ABB RobotStudio station: Solution3Working.rspag

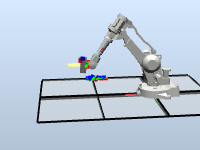
--- station ---
Station Solution3 (saved by RobotStudio 6.8.8307.1040)
Controller IRB_2400_12kg_1.55m
  mechanical unit ROB_1: IRB2400_10_150__02, 6 joints, base frame (0, 0, 0) mm
Layout (positions relative to the parent item):
  - IRB2400_10_150__02 [mechanism, from Robots\IRB2400_10_150_G_02.rslib] at (0, 0, 0) mm; joint values [0, 0.7222, 0.9922, 0, -0.9957, 0] (rad or m)
  - SickBox [smart component] at (1500, 0, 600) mm, rotated rx 0 ry -90 rz 0 deg
      properties: PointA=[1.29074548339844 0 0.569999938964844]; PointB=[1.28920959472656 0 0.6]; PointC=[1.29286682128906 0.0300000152587891 0.599999938964844]; Ax=1.29074548339844; Ay=0; Az=0.569999938964844; Bx=1.28920959472656; By=0; Bz=0.6; Cx=1.29286682128906; Cy=0.0300000152587891; Cz=0.599999938964844
      signals: AO Ax, AO Ay, AO Az, AO Bx, AO By, AO Bz, AO Cx, AO Cy, AO Cz
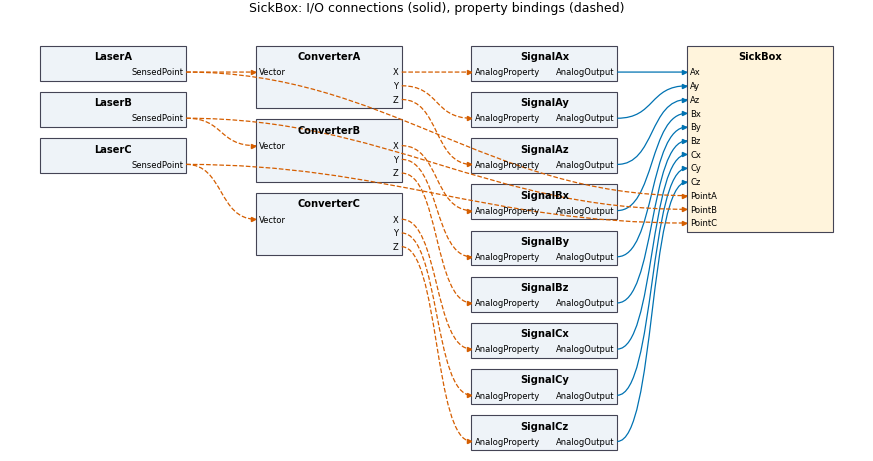
      connections:
        SignalAx.AnalogOutput -> SickBox.Ax
        SignalAy.AnalogOutput -> SickBox.Ay
        SignalAz.AnalogOutput -> SickBox.Az
        SignalBx.AnalogOutput -> SickBox.Bx
        SignalBy.AnalogOutput -> SickBox.By
        SignalBz.AnalogOutput -> SickBox.Bz
        SignalCx.AnalogOutput -> SickBox.Cx
        SignalCy.AnalogOutput -> SickBox.Cy
        SignalCz.AnalogOutput -> SickBox.Cz
        LaserA.SensedPoint => ConverterA.Vector
        LaserB.SensedPoint => ConverterB.Vector
        LaserC.SensedPoint => ConverterC.Vector
        LaserA.SensedPoint => SickBox.PointA
        LaserB.SensedPoint => SickBox.PointB
        LaserC.SensedPoint => SickBox.PointC
        ConverterA.X => SignalAx.AnalogProperty
        ConverterA.Y => SignalAy.AnalogProperty
        ConverterA.Z => SignalAz.AnalogProperty
        ConverterB.X => SignalBx.AnalogProperty
        ConverterB.Y => SignalBy.AnalogProperty
        ConverterB.Z => SignalBz.AnalogProperty
        ConverterC.X => SignalCx.AnalogProperty
        ConverterC.Y => SignalCy.AnalogProperty
        ConverterC.Z => SignalCz.AnalogProperty
    - LaserA [smart component, from Components\LineSensor.rslib]
        properties: Start=[-0.03 0 0]; End=[-0.03 0 0.3]; Radius=0.005; SensedPart=Brick; SensedPoint=[1.29074548339844 0 0.569999938964844]
      - _sensorPart_ [part]
    - LaserB [smart component, from Components\LineSensor.rslib]
        properties: Start=[0 0 0]; End=[0 0 0.3]; Radius=0.005; SensedPart=Brick; SensedPoint=[1.28920959472656 0 0.6]
      - _sensorPart_ [part]
    - LaserC [smart component, from Components\LineSensor.rslib] at (0, 30, 0) mm
        properties: Start=[0 0 0]; End=[0 0 0.3]; Radius=0.005; SensedPart=Brick; SensedPoint=[1.29286682128906 0.0300000152587891 0.599999938964844]
      - _sensorPart_ [part]
    - ConverterA [smart component, from Components\VectorConverter.rslib]
        properties: X=1.29074548339844; Y=0; Z=0.569999938964844; Vector=[1.29074548339844 0 0.569999938964844]
    - ConverterB [smart component, from Components\VectorConverter.rslib]
        properties: X=1.28920959472656; Y=0; Z=0.6; Vector=[1.28920959472656 0 0.6]
    - ConverterC [smart component, from Components\VectorConverter.rslib]
        properties: X=1.29286682128906; Y=0.0300000152587891; Z=0.599999938964844; Vector=[1.29286682128906 0.0300000152587891 0.599999938964844]
    - SignalAx [smart component, from Components\Converter.rslib]
        properties: AnalogProperty=1.29074548339844; DigitalProperty=0; BooleanProperty=false; GroupProperty=0
    - SignalAy [smart component, from Components\Converter.rslib]
        properties: AnalogProperty=0; DigitalProperty=0; BooleanProperty=false; GroupProperty=0
    - SignalAz [smart component, from Components\Converter.rslib]
        properties: AnalogProperty=0.569999938964844; DigitalProperty=0; BooleanProperty=false; GroupProperty=0
    - SignalBx [smart component, from Components\Converter.rslib]
        properties: AnalogProperty=1.28920959472656; DigitalProperty=0; BooleanProperty=false; GroupProperty=0
    - SignalBy [smart component, from Components\Converter.rslib]
        properties: AnalogProperty=0; DigitalProperty=0; BooleanProperty=false; GroupProperty=0
    - SignalBz [smart component, from Components\Converter.rslib]
        properties: AnalogProperty=0.6; DigitalProperty=0; BooleanProperty=false; GroupProperty=0
    - SignalCx [smart component, from Components\Converter.rslib]
        properties: AnalogProperty=1.29286682128906; DigitalProperty=0; BooleanProperty=false; GroupProperty=0
    - SignalCy [smart component, from Components\Converter.rslib]
        properties: AnalogProperty=0.0300000152587891; DigitalProperty=0; BooleanProperty=false; GroupProperty=0
    - SignalCz [smart component, from Components\Converter.rslib]
        properties: AnalogProperty=0.599999938964844; DigitalProperty=0; BooleanProperty=false; GroupProperty=0
  - RapidVariable [smart component, from Components\RapidVariable.rslib]
      properties: DataType=num; Controller=IRB_2400_12kg_1.55m; Task=T_ROB1; Module=Tests; Variable=TestVariable; Value=42.42
  - BrickPositioner [smart component]
      properties: GeneratedPart=(none)
      signals: DI DoMove, DI DoReset
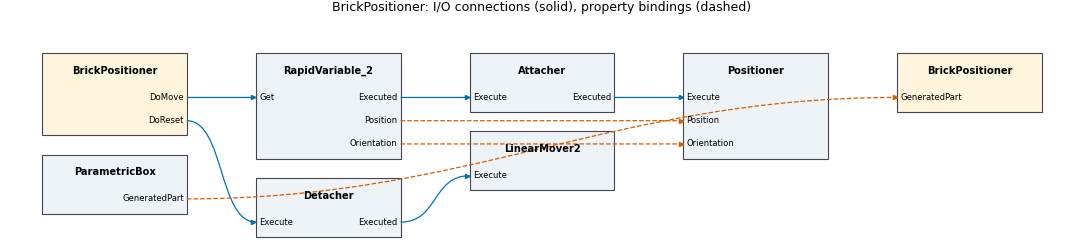
      connections:
        BrickPositioner.DoMove -> RapidVariable_2.Get
        RapidVariable_2.Executed -> Attacher.Execute
        Attacher.Executed -> Positioner.Execute
        BrickPositioner.DoReset -> Detacher.Execute
        Detacher.Executed -> LinearMover2.Execute
        RapidVariable_2.Position => Positioner.Position
        RapidVariable_2.Orientation => Positioner.Orientation
        ParametricBox.GeneratedPart => BrickPositioner.GeneratedPart
    - Positioner [smart component, from Components\Positioner.rslib]
        properties: Object=CalibBrick; Position=[1.29098 0.0609963 0.710539]; Orientation=[-2.29104981648406 1.49473022128042 0.730896849087735]; Reference=Global; ReferenceObject=(none)
    - RapidVariable_2 [smart component, from Components\RapidVariable.rslib]
        properties: DataType=pose; Controller=IRB_2400_12kg_1.55m; Task=T_ROB1; Module=Tests; Variable=BrickGlobal; Value=0; Position=[1.29098 0.0609963 0.710539]; Orientation=[-2.29104981648406 1.49473022128042 0.730896849087735]
    - Brick [part] at (1174.16, -75.63, 696.96) mm, rotated rx 48.15 ry 85.64 rz 41.28 deg
    - PositionSensor [smart component, from Components\PositionSensor.rslib]
        properties: Object=(none); Reference=Object; ReferenceObject=Brick; Position=[-4.78966566863637E-06 0.149996949808433 0.0999939037329676]; Orientation=[3.14140029990195 0.000646299912650163 0.000467407517623385]
    - Attacher [smart component, from Components\Attacher.rslib]
        properties: Parent=RapidVariable_2; Flange=0; Child=CalibBrick; Mount=false; Offset=[0 0 0]; Orientation=[0 0 0]
    - Detacher [smart component, from Components\Detacher.rslib]
        properties: Child=CalibBrick; KeepPosition=false
    - LinearMover2 [smart component, from Components\LinearMover2.rslib]
        properties: Object=CalibBrick; Direction=[0 1 0]; Distance=0.3; Duration=0.5; Reference=Global; ReferenceObject=(none)
  - CalibBrick [mechanism] at (1290.98, 61, 710.54) mm, rotated rx -131.27 ry 85.64 rz 41.88 deg
      TCP CalibBrickCorner at (0, 0, 0) mm
      links: CalibBrick
Attachment: Brick is attached to IRB2400_10_150__02 / Link6
Attachment: CalibBrick is attached to RapidVariable_2
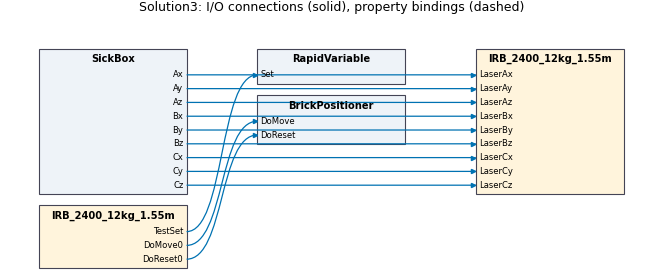
Station logic (signal -> signal, property => property):
  SickBox.Ax -> IRB_2400_12kg_1.55m.LaserAx
  IRB_2400_12kg_1.55m.TestSet -> RapidVariable.Set
  SickBox.Ay -> IRB_2400_12kg_1.55m.LaserAy
  SickBox.Az -> IRB_2400_12kg_1.55m.LaserAz
  SickBox.Bx -> IRB_2400_12kg_1.55m.LaserBx
  SickBox.By -> IRB_2400_12kg_1.55m.LaserBy
  SickBox.Bz -> IRB_2400_12kg_1.55m.LaserBz
  SickBox.Cx -> IRB_2400_12kg_1.55m.LaserCx
  SickBox.Cy -> IRB_2400_12kg_1.55m.LaserCy
  SickBox.Cz -> IRB_2400_12kg_1.55m.LaserCz
  IRB_2400_12kg_1.55m.DoMove0 -> BrickPositioner.DoMove
  IRB_2400_12kg_1.55m.DoReset0 -> BrickPositioner.DoReset
Targets, tools, work objects and paths stored in the station and not in the controller backup, written as RAPID:
! task T_ROB1
MODULE Module1
  CONST robtarget Target_70:=[[850.286116462,0,339.127587174],[0.708341194,0,0.70587021,0],[0,0,0,0],[9E+09,9E+09,9E+09,9E+09,9E+09,9E+09]];
ENDMODULE


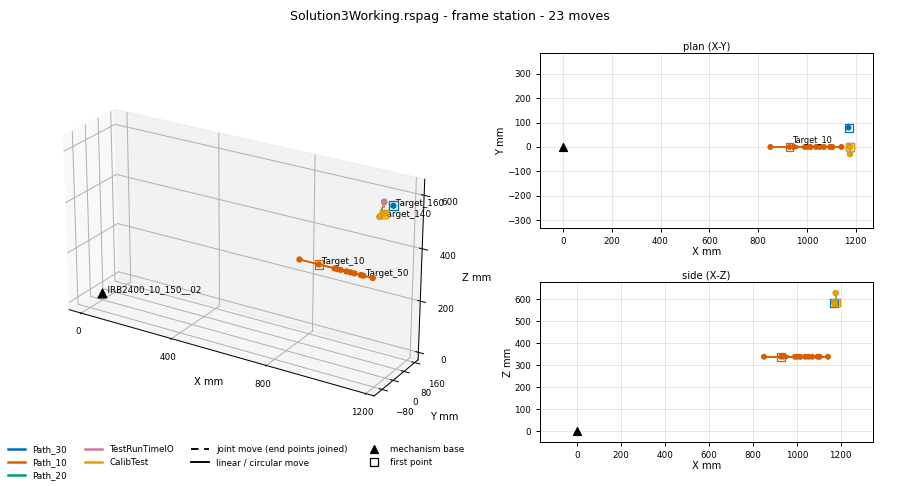
[picture p0: tool path of Solution3Working.rspag in frame station, 23 of 24 moves have a stored position in this frame; points joined in program order, loops and branches not executed]
--- Backups/IRB_2400_12kg_1.55m/RAPID/TASK1/PROGMOD/CalibData.mod ---
MODULE CalibData
	PERS tooldata CalibBrickCorner:=[TRUE,[[1290.98,60.9963,710.539],[0.0613583,-0.724242,0.0231326,0.686421]],[1,[131.249,-61.9822,-51.7883],[1,0,0,0],0,0,0]];
ENDMODULE

--- Backups/IRB_2400_12kg_1.55m/RAPID/TASK1/PROGMOD/Module1.mod ---
MODULE Module1

    PERS tooldata CalibratedBrick := [ TRUE, [[0, 0, 0], [1, 0, 0 ,0]], [5, [23, 0, 75], [1, 0, 0, 0], 0, 0, 0]];

    CONST robtarget Target_10:=[[928.612117607,0,339.127604265],[0.708341194,0,0.70587021,0],[0,0,0,0],[9E+09,9E+09,9E+09,9E+09,9E+09,9E+09]];
    CONST robtarget Target_20:=[[1002.038026848,0.000001175,339.127612489],[0.618553495,-0.20002778,0.758050904,-0.052338209],[-1,-1,-1,0],[9E+09,9E+09,9E+09,9E+09,9E+09,9E+09]];
    CONST robtarget Target_30:=[[1037.734049442,0.000005579,339.127592433],[0.642687352,0.413158989,0.644332092,0.032996567],[0,0,0,0],[9E+09,9E+09,9E+09,9E+09,9E+09,9E+09]];
    CONST robtarget Target_40:=[[1070.000069019,0.000006695,339.127578252],[0.232362667,-0.615252617,0.373665183,-0.654099488],[0,0,2,0],[9E+09,9E+09,9E+09,9E+09,9E+09,9E+09]];
    CONST robtarget Target_50:=[[1104.372000991,0.000002008,339.127566424],[0.775876893,-0.393805319,0.427062811,-0.246068635],[-1,-1,3,0],[9E+09,9E+09,9E+09,9E+09,9E+09,9E+09]];
    CONST robtarget Target_60:=[[1141.493005794,0.000005925,339.127521555],[0.523844629,0.121646721,0.777152572,-0.326837512],[0,0,3,0],[9E+09,9E+09,9E+09,9E+09,9E+09,9E+09]];

    CONST pos baseA := [10,1,1];
    CONST pos dirA := [-1,0,0];
    CONST pos baseB := [10,0,1];
    CONST pos dirB := [-1,0,0];
    CONST pos baseC := [10,1,0];
    CONST pos dirC := [-1,0,0];

    !LaserCalib -> hardcode kalibration values
    CONST pos laserA0 := [1690,10,670];
    CONST pos laserA1 := [-1,0,0];
    CONST pos laserB0 := [1690,0,670];
    CONST pos laserB1 := [-1,0,0];
    CONST pos laserC0 := [1690,10,680];
    CONST pos laserC1 := [-1,0,0];

    CONST num array{4} := [1,2,3,4];
    VAR num testarray{4}:=array;
    VAR num plane{4}:=[0,0,0,0];
    CONST robtarget Target_80:=[[850.286116462,0,339.127587174],[0.708341194,0,0.70587021,0],[0,0,0,0],[9E+09,9E+09,9E+09,9E+09,9E+09,9E+09]];
    CONST robtarget Target_90:=[[1094.704044152,0.000007314,339.12751907],[0.616775815,-0.341477844,0.708630274,0.028698629],[-1,-1,3,0],[9E+09,9E+09,9E+09,9E+09,9E+09,9E+09]];
    CONST robtarget Target_100:=[[1053.23509452,0.000003121,339.127514541],[0.869733098,0.028795386,0.474790845,0.131562978],[-1,-1,4,0],[9E+09,9E+09,9E+09,9E+09,9E+09,9E+09]];
    CONST robtarget Target_110:=[[1015.094978375,0.000003488,339.127487816],[0.550234045,-0.282952574,0.59944613,-0.507784081],[0,0,3,0],[9E+09,9E+09,9E+09,9E+09,9E+09,9E+09]];
    CONST robtarget Target_120:=[[991.513733063,0.000004798,339.127497052],[0.365097325,-0.7846233,0.391266315,-0.313018995],[-1,-1,2,0],[9E+09,9E+09,9E+09,9E+09,9E+09,9E+09]];
    CONST robtarget Target_130:=[[1176.9139888,0.000006322,586.026163881],[0.708341005,-0.000000414,0.7058704,-0.00000011],[-1,-1,-1,0],[9E+09,9E+09,9E+09,9E+09,9E+09,9E+09]];
    CONST robtarget Target_140:=[[1176.913999337,-29.620214443,586.026196841],[0.490684914,-0.509075862,0.488973111,0.510857494],[-1,-2,0,0],[9E+09,9E+09,9E+09,9E+09,9E+09,9E+09]];
    CONST robtarget Target_150:=[[1176.913967292,0.000006322,629.779686498],[0.001946977,0.00000037,-0.999998105,-0.000000216],[-1,0,-1,0],[9E+09,9E+09,9E+09,9E+09,9E+09,9E+09]];

    CONST pos LaserPtsOnBrick{9} := [[1276.97, 0.00, 570.00],[1276.87, 0.00, 600.00],[1276.87, 30.00, 600.00],[1251.10, 0.00, 570.00],[1251.10, 0.00, 600.00],[1249.89, 30.00, 600.00],[1282.30, 0.00, 570.00],[1282.42, 0.00, 600.00],[1282.42, 30.00, 600.00]];
    CONST pose TestPose := [Target_130.trans, Target_130.rot];
    CONST pos TestOffset := [10, 10, 10];
    CONST pos TestPos := TestPose.trans+TestOffset;
    VAR pose inv;
    CONST robtarget Target_160:=[[1170.892026522,78.961400265,586.005220528],[0.519569231,0.481450787,0.517756592,-0.479771888],[0,1,-1,0],[9E+09,9E+09,9E+09,9E+09,9E+09,9E+09]];

    PROC main()
        !Path_30;
        !Path_10;
        !CalibTest;
        !Path_20;
        !WritePosArray(LaserPtsOnBrick);
        !TestPoseVect;
        !PlanesTest;
        !IDunno;
        !TestMatrixSolve;
        !TestIO;
        !TestRunTimeIO;
        TestSimCalib;
    ENDPROC


     FUNC string ArrayToString(num array{*})
        VAR string s := "[ ";
        FOR i FROM 1 TO DIM(array,1) DO
            s := s + ValToStr(array{i});
            s := s + " ";
        ENDFOR
        s := s + "]";
        RETURN s;
    ENDFUNC

    PROC WritePosArray(pos array{*})
        FOR i FROM 1 TO DIM(array,1) DO
            TPWrite "Tool pos: " \Pos:=array{i};
        ENDFOR
    ENDPROC

    FUNC string WritePlaneArray(num array{*})
        VAR string s;
        s:="";
        s:=s+"[";
        FOR i FROM 1 TO DIM(array,1) DO
            s:=s+" ";
            s:= s + NumToStr(array{i}, 4);
        ENDFOR
        s:=s+"]";
        RETURN s;
    ENDFUNC

    PROC Path_30()
        MoveL Target_160,v1000,z100,tool0\WObj:=wobj0;
    ENDPROC



    !Proc for (pos1, pos2, pos3) -> plane (flange)

    !Proc (plan1, plan2, plan3) -> origo & 3 coordiante axies

    !Proc (origo, x-axis, y-axis, z-axis) (flange) -> tooldata






ENDMODULE

--- Backups/IRB_2400_12kg_1.55m/RAPID/TASK1/PROGMOD/Paths.mod ---
MODULE Paths

    PROC Path_10()
        TPErase;
        MoveL Target_10,v1000,z100,tool0\WObj:=wobj0;
        MoveL Target_20,v1000,z100,tool0\WObj:=wobj0;
        MoveL Target_30,v1000,z100,tool0\WObj:=wobj0;
        MoveL Target_40,v1000,z100,tool0\WObj:=wobj0;
        MoveL Target_50,v1000,z100,tool0\WObj:=wobj0;
        MoveL Target_60,v1000,z100,tool0\WObj:=wobj0;
        MoveL Target_80,v1000,z100,tool0\WObj:=wobj0;
        MoveL Target_90,v1000,z100,tool0\WObj:=wobj0;
        MoveL Target_100,v1000,z100,tool0\WObj:=wobj0;
        MoveL Target_110,v1000,z100,tool0\WObj:=wobj0;
        MoveL Target_120,v1000,z100,tool0\WObj:=wobj0;
    ENDPROC

    PROC Path_20()
        MoveL Target_130,v1000,z100,tool0\WObj:=wobj0;
        MoveL Target_140,v1000,z100,tool0\WObj:=wobj0;
        MoveL Target_150,v1000,z100,tool0\WObj:=wobj0;
    ENDPROC
ENDMODULE

--- Backups/IRB_2400_12kg_1.55m/RAPID/TASK1/PROGMOD/Tests.mod ---
MODULE Tests

    VAR num TestVariable;
    VAR robtarget corner := [[1015.094978375,0.000003488,339.127487816],[0.550234045,-0.282952574,0.59944613,-0.507784081],[0,0,3,0],[9E+09,9E+09,9E+09,9E+09,9E+09,9E+09]];
    VAR pose BrickGlobal;

    PROC TestSimCalib()

        VAR pos BrickPoints{3,3};
        VAR robtarget CalibPath{4}:=[Target_130,Target_160,Target_150,Target_130];
        VAR robtarget t;
        VAR pos nTop;
        VAR pos nSide;
        VAR pos nFront;
        VAR num Top{4};
        VAR num Side{4};
        VAR num Front{4};
        VAR num M{3,4};
        VAR pos orig;
        VAR pos xDir;
        VAR pos yDir;
        VAR pos zDir;
        VAR pose BrickCornerLocal;
        VAR pose ToolLocal;
        VAR pose BrickCornerGlobal;
        PulseDO DoReset0;
        FOR targ FROM 1 TO 4 DO
            MoveJ CalibPath{targ},v100,fine,tool0\WObj:=wobj0;
            WaitTime 1.5;
            IF targ<4 THEN
                BrickPoints{targ,1}:=InToolFrame(ReadSimLaser("A"));
                BrickPoints{targ,2}:=InToolFrame(ReadSimLaser("B"));
                BrickPoints{targ,3}:=InToolFrame(ReadSimLaser("C"));
            ENDIF
            WaitTime 1.0;
        ENDFOR
        CalcPlane BrickPoints{1,1},BrickPoints{1,2},BrickPoints{1,3},Top;
        CalcPlane BrickPoints{2,1},BrickPoints{2,2},BrickPoints{2,3},Side;
        CalcPlane BrickPoints{3,1},BrickPoints{3,2},BrickPoints{3,3},Front;
        FOR j FROM 1 TO 4 DO
            M{1,j}:=Top{j};
            M{2,j}:=Side{j};
            M{3,j}:=Front{j};
        ENDFOR
        TPWrite "-----------OLD-----------";
        TPWrite "Old tool pos: " \Pos:=CalibBrickCorner.tframe.trans;
        TPWrite "Old tool rot: " \Orient:=CalibBrickCorner.tframe.rot;
        orig:=SolvePlanes(M);
        nTop:=[Top{1},Top{2},Top{3}];
        nSide:=[Side{1},Side{2},Side{3}];
        nFront:=[Front{1},Front{2},Front{3}];
        xDir:=RoundPos(NormalizePos(CrossProd(nSide,nTop)),4);
        yDir:=RoundPos(NormalizePos(CrossProd(nTop,nFront)),4);
        zDir:=RoundPos(NormalizePos(CrossProd(nFront,nSide)),4);
        BrickCornerLocal:=[orig,MakeQuaternions(xDir,yDir,zDir)];
        t:=CRobT(\Tool:=tool0 \WObj:=wobj0);
        ToolLocal:=[t.trans,t.rot];
        BrickCornerGlobal:=PoseMult(ToolLocal,BrickCornerLocal);
        BrickGlobal:=BrickCornerGlobal;
        !TPErase;
        TPWrite "----------CALC------------";
        TPWrite "BrickCornerGlobal.trans: " \Pos:=BrickCornerGlobal.trans;
        TPWrite "BrickCornerGlobal.rot: " \Orient:=BrickCornerGlobal.rot;

        !corner := [BrickCornerGlobal.trans,BrickCornerGlobal.rot,[0,0,0,0],[9E+09,9E+09,9E+09,9E+09,9E+09,9E+09]]
        PulseDO DoMove0;
        CalibBrickCorner.tframe:=BrickCornerGlobal;
        TPWrite "---------NEW-------------";
        TPWrite "New tool pos: " \Pos:=CalibBrickCorner.tframe.trans;
        TPWrite "New tool rot: " \Orient:=CalibBrickCorner.tframe.rot;
    ENDPROC

    PROC TestRunTimeIO()
        TPErase;
        MoveJ Target_130,v100,fine,tool0\WObj:=wobj0;
        WaitTime 2.0;
        TPWrite "------------";
        TestIO;
        WaitTime 2.0;
        MoveJ Target_140,v100,fine,tool0\WObj:=wobj0;
        WaitTime 2.0;
        TPWrite "------------";
        TestIO;
        WaitTime 2.0;
        MoveJ Target_150,v100,fine,tool0\WObj:=wobj0;
        WaitTime 2.0;
        TPWrite "------------";
        TestIO;
        WaitTime 2.0;
        MoveJ Target_130,v100,z100,tool0\WObj:=wobj0;
        TPWrite "------------";
        WaitTime 1.0;
    ENDPROC

    PROC TestIO()
        !TPErase;
        !TPWrite "TestVariable: " \Num:=TestVariable;
        TPWrite "LaserA Global: " \Pos:=ReadSimLaser("A");
        TPWrite "LaserA Tool: " \Pos:=InToolFrame(ReadSimLaser("A"));
        TPWrite "LaserB Global: " \Pos:=ReadSimLaser("B");
        TPWrite "LaserB Tool: " \Pos:=InToolFrame(ReadSimLaser("B"));
        TPWrite "LaserC Global: " \Pos:=ReadSimLaser("C");
        TPWrite "LaserC Tool: " \Pos:=InToolFrame(ReadSimLaser("C"));
    ENDPROC

    PROC TestPoseVect()
        TPErase;
        TPWrite "TestPos: " \Pos:=TestPos;
        TPWrite "TestPose.trans: " \Pos:=TestPose.trans;
        TPWrite "TestPos.rot: " \Orient:=TestPose.rot;
        TPWrite "PoseVect(TestPose, TestOffset): " \Pos:=PoseVect(TestPose, TestOffset);
        inv := PoseInv(TestPose);
        TPWrite "PoseInv.trans: " \Pos:=inv.trans;
        TPWrite "PoseInv.rot: " \Orient:=inv.rot;
        TPWrite "PoseVect(inv, TestOffset): " \Pos:=PoseVect(inv, TestOffset);
        TPWrite "------------";
        TPWrite "PoseVect(TestPose, TestPos): " \Pos:=PoseVect(TestPose, TestPos);
        TPWrite "PoseVect(inv, TestPos): " \Pos:=PoseVect(inv, TestPos);
    ENDPROC

    PROC TestMatrixSolve()
        CONST dnum M{3,3}:=[[1,1,1],[1,0,-1],[-2,1,0]];
        CONST dnum d{3}:=[13,-2,3];
        VAR dnum x{3};
        VAR pos p;
        MatrixSolve M, d, x;
        p:=[DnumToNum(x{1}), DnumToNum(x{2}), DnumToNum(x{3})];
        TPErase;
        TPWrite "test: " \Pos:=p;
    ENDPROC

    PROC PlanesTest()
        VAR pos BrickPoints{9};
        VAR robtarget targs{9}:=[Target_130,Target_130,Target_130,Target_140,Target_140,Target_140,Target_150,Target_150,Target_150];
        VAR pos nTop;
        VAR pos nSide;
        VAR pos nFront;
        VAR num Top{4};
        VAR num Side{4};
        VAR num Front{4};
        VAR num M{3,4};
        VAR pos orig;
        VAR pos xDir;
        VAR pos yDir;
        VAR pos zDir;
        FOR i FROM 1 TO 9 DO
            BrickPoints{i}:=InToolFrameHardcode(LaserPtsOnBrick{i}, targs{i});
        ENDFOR
        TPErase;
        CalcPlane BrickPoints{1},BrickPoints{2},BrickPoints{3},Top;
        CalcPlane BrickPoints{4},BrickPoints{5},BrickPoints{6},Side;
        CalcPlane BrickPoints{7},BrickPoints{8},BrickPoints{9},Front;
        FOR j FROM 1 TO 4 DO
            M{1,j}:=Top{j};
            M{2,j}:=Side{j};
            M{3,j}:=Front{j};
        ENDFOR
        orig:=SolvePlanes(M);
        nTop:=[Top{1},Top{2},Top{3}];
        nSide:=[Side{1},Side{2},Side{3}];
        nFront:=[Front{1},Front{2},Front{3}];


        TPWrite "orig: " \Pos:=orig;
        TPWrite "xDir: " \Pos:=RoundPos(NormalizePos(CrossProd(nTop,nSide)),4);
        TPWrite "yDir: " \Pos:=RoundPos(NormalizePos(CrossProd(nFront,nTop)),4);
        TPWrite "zDir: " \Pos:=RoundPos(NormalizePos(CrossProd(nFront,nSide)),4);
    ENDPROC

    PROC CalibTest()
        TPErase;
        MoveJ Target_130,v100,fine,tool0\WObj:=wobj0;
        WaitTime 2.0;
        TPWrite "------------";
        !TPWrite "Global pos: " \Pos:=LaserPtsOnBrick{1};
        TPWrite "Tool pos: " \Pos:=InToolFrame(LaserPtsOnBrick{1});
        !TPWrite "Global pos: " \Pos:=LaserPtsOnBrick{2};
        TPWrite "Tool pos: " \Pos:=InToolFrame(LaserPtsOnBrick{2});
        !TPWrite "Global pos: " \Pos:=LaserPtsOnBrick{3};
        TPWrite "Tool pos: " \Pos:=InToolFrame(LaserPtsOnBrick{3});
        WaitTime 2.0;
        MoveJ Target_140,v100,fine,tool0\WObj:=wobj0;
        WaitTime 2.0;
        TPWrite "------------";
        !TPWrite "Global pos: " \Pos:=LaserPtsOnBrick{4};
        TPWrite "Tool pos: " \Pos:=InToolFrame(LaserPtsOnBrick{4});
        !TPWrite "Global pos: " \Pos:=LaserPtsOnBrick{5};
        TPWrite "Tool pos: " \Pos:=InToolFrame(LaserPtsOnBrick{5});
        !TPWrite "Global pos: " \Pos:=LaserPtsOnBrick{6};
        TPWrite "Tool pos: " \Pos:=InToolFrame(LaserPtsOnBrick{6});
        WaitTime 2.0;
        MoveJ Target_150,v100,fine,tool0\WObj:=wobj0;
        WaitTime 2.0;
        TPWrite "------------";
        !TPWrite "Global pos: " \Pos:=LaserPtsOnBrick{7};
        TPWrite "Tool pos: " \Pos:=InToolFrame(LaserPtsOnBrick{7});
        !TPWrite "Global pos: " \Pos:=LaserPtsOnBrick{8};
        TPWrite "Tool pos: " \Pos:=InToolFrame(LaserPtsOnBrick{8});
        !TPWrite "Global pos: " \Pos:=LaserPtsOnBrick{9};
        TPWrite "Tool pos: " \Pos:=InToolFrame(LaserPtsOnBrick{9});
        WaitTime 2.0;
        MoveJ Target_130,v100,z100,tool0\WObj:=wobj0;
        TPWrite "------------";
        WaitTime 1.0;

    ENDPROC




ENDMODULE

--- Backups/IRB_2400_12kg_1.55m/RAPID/TASK1/SYSMOD/LinAlgRoutines.sys ---
MODULE LinAlgRoutines(SYSMODULE)


    !Procedure to calculate the equation of the plane through the three given points
    !   IN pos p1, p2, p3 & empty num array plane{4}
    !   OUT num plane{4} will contain a, b, c, d for equation: ax+by+cz=d
    PROC CalcPlane(pos p1, pos p2, pos p3, INOUT num plane{*})
        VAR pos v1;
        VAR pos v2;
        VAR pos normal;
        VAR num d;
        v1:=p2-p1;
        v2:=p3-p1;
        normal:= CrossProd(v1,v2);
        d:= DotProd(normal, p1);
        plane{1}:=normal.x;
        plane{2}:=normal.y;
        plane{3}:=normal.z;
        plane{4}:=d;
    ENDPROC

    !Proc for laser_value -> pos (bas)
    FUNC pos LaserCoordinate(num k, pos base, pos dir)
        RETURN k*dir+base;
    ENDFUNC

    !Function to translate a given point (pos p) into a point in the flange frame
    FUNC pos InToolFrame(pos p)
        !The current position of the robot's flange as a robtarget
        VAR robtarget Targ;
        !The current position of the robot's flange as a pose.
        !   pose <=> linear transformation from local coordiantes -> global coordinates
        VAR pose Flange;
        !The inverse transformation of the flange
        !   global coordinates -> flange coordinates
        VAR pose InvFlange;
        !assign values
        Targ:=CRobT(\Tool:=tool0 \WObj:=wobj0);
        Flange:=[Targ.trans,Targ.rot];
        InvFlange:=PoseInv(Flange);
        !return the pos p transformed from global -> flange coordinates
        RETURN PoseVect(InvFlange,p);
    ENDFUNC

    FUNC pos InToolFrameHardcode(pos p, robtarget Targ)
        VAR pose Flange;
        VAR pose InvFlange;
        Flange:=[Targ.trans,Targ.rot];
        InvFlange:=PoseInv(Flange);
        RETURN PoseVect(InvFlange,p);
    ENDFUNC

    FUNC pos SolvePlanes(num matrix{*,*})
        VAR dnum M{3,3};
        VAR dnum d{3};
        VAR dnum x{3};
        VAR pos p;
        FOR i FROM 1 TO 3 DO
            FOR j FROM 1 TO 3 DO
                M{i,j}:=NumToDnum(matrix{i,j});
            ENDFOR
            d{i}:=NumToDnum(matrix{i,4});
        ENDFOR
        MatrixSolve M, d, x;
        p:=[DnumToNum(x{1}),DnumToNum(x{2}),DnumToNum(x{3})];
        RETURN p;
    ENDFUNC


    FUNC pos RoundPos(pos p, num dec)
        p.x:= Round(p.x \Dec:=dec);
        p.y:= Round(p.y \Dec:=dec);
        p.z:= Round(p.z \Dec:=dec);
        RETURN p;
    ENDFUNC

    FUNC pos NormalizePos(pos p)
        VAR num pn;
        pn:=sqrt(p.x*p.x+p.y*p.y+p.z*p.z);
        p.x:=p.x/pn;
        p.y:=p.y/pn;
        p.z:=p.z/pn;
        RETURN p;
    ENDFUNC

    FUNC orient MakeQuaternions(pos x, pos y, pos z)
        VAR num q1;
        VAR num q2;
        VAR num q3;
        VAR num q4;
        VAR num sign2:=1;
        VAR num sign3:=1;
        VAR num sign4:=1;
        VAR orient q;
        IF y.z-z.y<0 THEN
            sign2:=-1;
        ENDIF
        IF z.x-x.z<0 THEN
            sign3:=-1;
        ENDIF
        IF x.y-y.x<0 THEN
            sign4:=-1;
        ENDIF
        q1:=sqrt(x.x+y.y+z.z+1)/2;
        q2:=sqrt(x.x-y.y-z.z+1)/2*sign2;
        q3:=sqrt(y.y-x.x-z.z+1)/2*sign3;
        q4:=sqrt(z.z-x.x-y.y+1)/2*sign4;

        q:=[q1,q2,q3,q4];
        RETURN NOrient(q);
    ENDFUNC

    FUNC pos ReadSimLaser(string laser)
        CONST num k:=1000;
        VAR pos p;
        TEST laser
        CASE "A":p:=[AInput(LaserAx)*k, AInput(LaserAy)*k, AInput(LaserAz)*k];
        CASE "B":p:=[AInput(LaserBx)*k, AInput(LaserBy)*k, AInput(LaserBz)*k];
        CASE "C":p:=[AInput(LaserCx)*k, AInput(LaserCy)*k, AInput(LaserCz)*k];
        DEFAULT:p:=[0,0,0];
        ENDTEST

        RETURN p;
    ENDFUNC


ENDMODULE

--- Backups/IRB_2400_12kg_1.55m/SYSPAR/EIO.cfg ---
EIO:CFG_1.0:6:1::
#
EIO_SIGNAL:

      -Name "LaserAx" -SignalType "AI" -Access "All" -MaxLog 20 -MinLog -20

      -Name "TestInput" -SignalType "AI" -Access "All"

      -Name "TestDigInput0" -SignalType "DI" -Access "All"

      -Name "TestSet" -SignalType "DO" -Access "All"

      -Name "LaserAy" -SignalType "AI" -Access "All"

      -Name "LaserAz" -SignalType "AI" -Access "All"

      -Name "LaserBx" -SignalType "AI" -Access "All"

      -Name "LaserBy" -SignalType "AI" -Access "All"

      -Name "LaserBz" -SignalType "AI" -Access "All"

      -Name "LaserCx" -SignalType "AI" -Access "All"

      -Name "LaserCy" -SignalType "AI" -Access "All"

      -Name "LaserCz" -SignalType "AI" -Access "All"

      -Name "DoMove0" -SignalType "DO" -Access "All"

      -Name "DoReset0" -SignalType "DO" -Access "All"
